TYPE StringHandle_t : POINTER TO STRING(255); END_TYPE

(* stored: Version 1.1.0.1, ProductVersion 3.1.4022.9
   DUT StringHandle_t: Id {b00b16aa-a1c0-41cd-9b04-c61a581ed61c} *)
